// TIA Portal V15.1 export
// export: Created 2024-06-21T08:41:12.3335772Z, ExportSetting WithDefaults, DisplayName Totally Integrated Automation Portal, DisplayVersion V15.1 Update 5, DisplayName TIA Portal Openness, DisplayVersion V15.1 Update 5, DisplayName SINAMICS Startdrive Advanced, DisplayVersion V15.1, DisplayName G130, G150, S120, S150, SINAMICS MV, S210, DisplayVersion V15.1, DisplayName G110M, G120, G120C, G120D, G120P, DisplayVersion V15.1, DisplayName STEP 7 Professional, DisplayVersion V15.1 Update 5, DisplayName STEP 7 Safety, DisplayVersion V15.1, DisplayName WinCC Professional, DisplayVersion V15.1 Update 5, DisplayName SIMATIC Visualization Architect, DisplayVersion V15.1
FUNCTION_BLOCK "LGBHMILed"   // FB6683, FBD
TITLE = LGBHMILed
{ S7_Optimized_Access := 'TRUE' }
VERSION : 0.1
// =============================================================================
// This module handles indication for Start, Alarm Reset.
// =============================================================================
// stored: AutoNumber false, IsIECCheckEnabled false, IsRetainMemResEnabled false, MemoryReserve 100, SetENOAutomatically False, UDAEnableTagReadback false
   VAR_INPUT
      I_SafetyAckReq { ExternalAccessible := 'False'; ExternalVisible := 'False'; ExternalWritable := 'False'} : Bool;   // Safety acknowledge required
      I_SafetyOk { ExternalAccessible := 'False'; ExternalVisible := 'False'; ExternalWritable := 'False'} : Bool;   // All Safety ok
      I_PowerOnReq { ExternalAccessible := 'False'; ExternalVisible := 'False'; ExternalWritable := 'False'} : Bool;   // Request for power on (fast blinking of blue lamp)
      I_ResetSafety { ExternalAccessible := 'False'; ExternalVisible := 'False'; ExternalWritable := 'False'} : Bool;   // Reset Safety Signal of the Safety Zone
      C_ZSLevel { ExternalAccessible := 'False'; ExternalVisible := 'False'; ExternalWritable := 'False'} : Bool;   // ZS level OP
      C_PLCLevel { ExternalAccessible := 'False'; ExternalVisible := 'False'; ExternalWritable := 'False'} : Bool;   // PLC level OP
   END_VAR
   VAR_OUTPUT
      O_StartPBInd { ExternalAccessible := 'False'; ExternalVisible := 'False'; ExternalWritable := 'False'} : Bool;   // Start PB indication
      O_AlarmResetPBInd { ExternalAccessible := 'False'; ExternalVisible := 'False'; ExternalWritable := 'False'} : Bool;   // Alarm Reset PB Indication
   END_VAR
   VAR_IN_OUT
      IO_ModesZM1 : "Modes";   // Modes ZM1
      IO_ModesZM2 : "Modes";   // Modes ZM2
      IO_ModesZM3 : "Modes";   // Modes ZM3
      IO_ModesZM4 : "Modes";   // Modes ZM4
      IO_ModesZM5 : "Modes";   // Modes ZM5
      IO_ModesZM6 : "Modes";   // Modes ZM6
      IO_ModesZM7 : "Modes";   // Modes ZM7
      IO_ModesZM8 : "Modes";   // Modes ZM8
      IO_ModesZM9 : "Modes";   // Modes ZM9
      IO_ModesZM10 : "Modes";   // Modes ZM10
      IO_ModesZM11 : "Modes";   // Modes ZM11
      IO_ModesZM12 : "Modes";   // Modes ZM12
      IO_ModesZM13 : "Modes";   // Modes ZM13
      IO_ModesZM14 : "Modes";   // Modes ZM14
      IO_ModesZM15 : "Modes";   // Modes ZM15
      IO_ModesZM16 : "Modes";   // Modes ZM16
   END_VAR
   VAR
      ZMAlarmABLampSteadyCondition { ExternalAccessible := 'False'; ExternalVisible := 'False'; ExternalWritable := 'False'} : Bool;   // Alarm conditions active
      ZSAlarmABLampSteadyCondition { ExternalAccessible := 'False'; ExternalVisible := 'False'; ExternalWritable := 'False'} : Bool;   // Alarm conditions active
      PLCAlarmABLampSteadyCondition { ExternalAccessible := 'False'; ExternalVisible := 'False'; ExternalWritable := 'False'} : Bool;   // Alarm conditions active
      ZMAlarmABAckReq { ExternalAccessible := 'False'; ExternalVisible := 'False'; ExternalWritable := 'False'} : Bool;   // Alarm AB acknowledgement required
      ZSAlarmABAckReq { ExternalAccessible := 'False'; ExternalVisible := 'False'; ExternalWritable := 'False'} : Bool;   // Alarm AB acknowledgement required
      PLCAlarmABAckReq { ExternalAccessible := 'False'; ExternalVisible := 'False'; ExternalWritable := 'False'} : Bool;   // Alarm AB acknowledgement required
      BlueLampBlinkingCond { ExternalAccessible := 'False'; ExternalVisible := 'False'; ExternalWritable := 'False'} : Bool;   // Blue lamp blinking condition
      Lamptest { ExternalAccessible := 'False'; ExternalVisible := 'False'; ExternalWritable := 'False'} : Bool;   // Lamptest selected alternating signal
      LamptestSteady { ExternalAccessible := 'False'; ExternalVisible := 'False'; ExternalWritable := 'False'} : Bool;   // Lamptest selected steady signal
      AutoSel { ExternalAccessible := 'False'; ExternalVisible := 'False'; ExternalWritable := 'False'} : Bool;   // Automatic mode selected
      AutoMode { ExternalAccessible := 'False'; ExternalVisible := 'False'; ExternalWritable := 'False'} : Bool;   // Automatic mode active
      StartPBInd { ExternalAccessible := 'False'; ExternalVisible := 'False'; ExternalWritable := 'False'} : Bool;   // Start PB indication
      AlarmResetPBInd { ExternalAccessible := 'False'; ExternalVisible := 'False'; ExternalWritable := 'False'} : Bool;   // Alarm Reset PB Indication
   END_VAR
BEGIN

REGION Network 1: **** 4.2 - Machine status - Calculated **** ZM level Alarm condition AB active
   // Alarm condition AB active
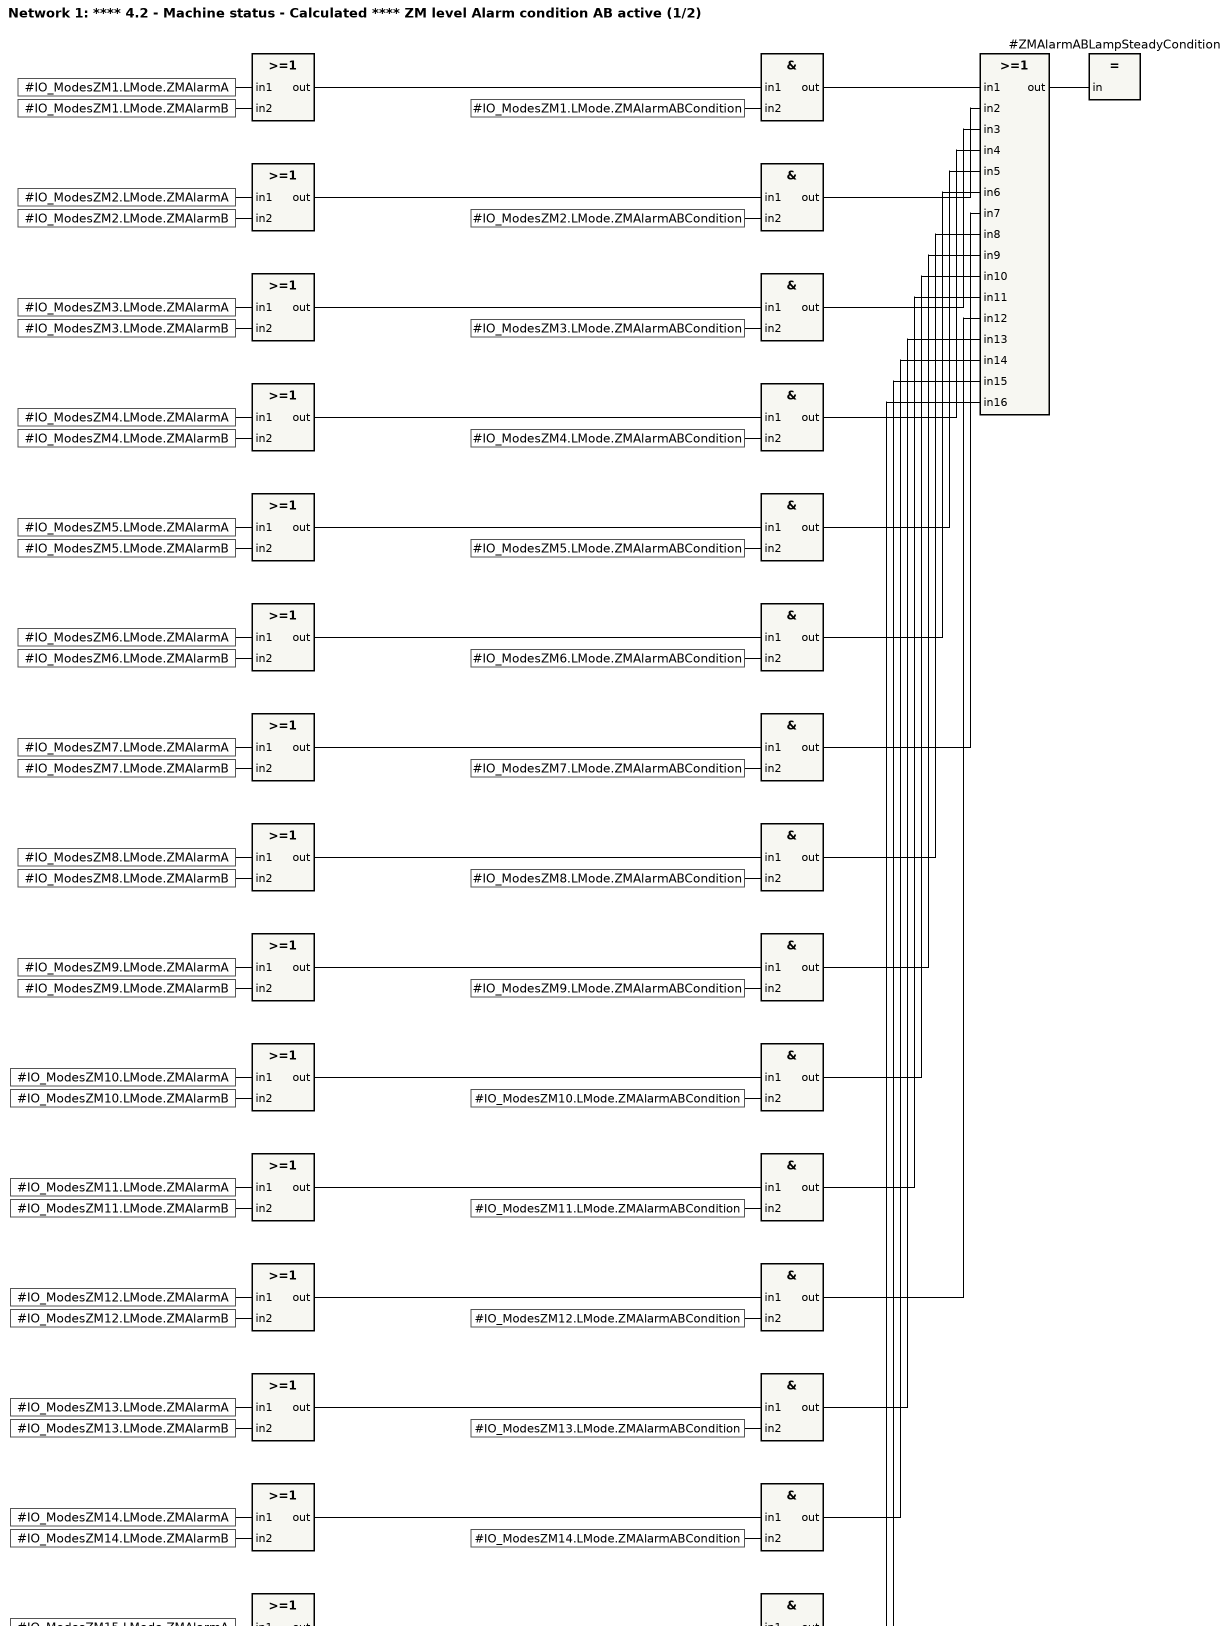
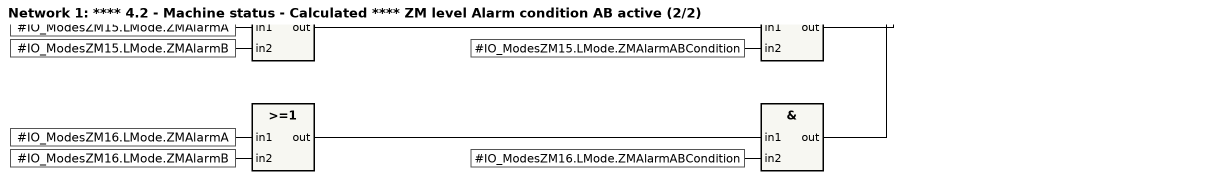
   #ZMAlarmABLampSteadyCondition := ((#IO_ModesZM1.LMode.ZMAlarmA OR #IO_ModesZM1.LMode.ZMAlarmB) AND #IO_ModesZM1.LMode.ZMAlarmABCondition) OR ((#IO_ModesZM2.LMode.ZMAlarmA OR #IO_ModesZM2.LMode.ZMAlarmB) AND #IO_ModesZM2.LMode.ZMAlarmABCondition) OR ((#IO_ModesZM3.LMode.ZMAlarmA OR #IO_ModesZM3.LMode.ZMAlarmB) AND #IO_ModesZM3.LMode.ZMAlarmABCondition) OR ((#IO_ModesZM4.LMode.ZMAlarmA OR #IO_ModesZM4.LMode.ZMAlarmB) AND #IO_ModesZM4.LMode.ZMAlarmABCondition) OR ((#IO_ModesZM5.LMode.ZMAlarmA OR #IO_ModesZM5.LMode.ZMAlarmB) AND #IO_ModesZM5.LMode.ZMAlarmABCondition) OR ((#IO_ModesZM6.LMode.ZMAlarmA OR #IO_ModesZM6.LMode.ZMAlarmB) AND #IO_ModesZM6.LMode.ZMAlarmABCondition) OR ((#IO_ModesZM7.LMode.ZMAlarmA OR #IO_ModesZM7.LMode.ZMAlarmB) AND #IO_ModesZM7.LMode.ZMAlarmABCondition) OR ((#IO_ModesZM8.LMode.ZMAlarmA OR #IO_ModesZM8.LMode.ZMAlarmB) AND #IO_ModesZM8.LMode.ZMAlarmABCondition) OR ((#IO_ModesZM9.LMode.ZMAlarmA OR #IO_ModesZM9.LMode.ZMAlarmB) AND #IO_ModesZM9.LMode.ZMAlarmABCondition) OR ((#IO_ModesZM10.LMode.ZMAlarmA OR #IO_ModesZM10.LMode.ZMAlarmB) AND #IO_ModesZM10.LMode.ZMAlarmABCondition) OR ((#IO_ModesZM11.LMode.ZMAlarmA OR #IO_ModesZM11.LMode.ZMAlarmB) AND #IO_ModesZM11.LMode.ZMAlarmABCondition) OR ((#IO_ModesZM12.LMode.ZMAlarmA OR #IO_ModesZM12.LMode.ZMAlarmB) AND #IO_ModesZM12.LMode.ZMAlarmABCondition) OR ((#IO_ModesZM13.LMode.ZMAlarmA OR #IO_ModesZM13.LMode.ZMAlarmB) AND #IO_ModesZM13.LMode.ZMAlarmABCondition) OR ((#IO_ModesZM14.LMode.ZMAlarmA OR #IO_ModesZM14.LMode.ZMAlarmB) AND #IO_ModesZM14.LMode.ZMAlarmABCondition) OR ((#IO_ModesZM15.LMode.ZMAlarmA OR #IO_ModesZM15.LMode.ZMAlarmB) AND #IO_ModesZM15.LMode.ZMAlarmABCondition) OR ((#IO_ModesZM16.LMode.ZMAlarmA OR #IO_ModesZM16.LMode.ZMAlarmB) AND #IO_ModesZM16.LMode.ZMAlarmABCondition);
END_REGION

REGION Network 2: **** 4.2 - Machine status - Calculated **** ZS level Alarm condition AB active
   // Alarm condition AB active
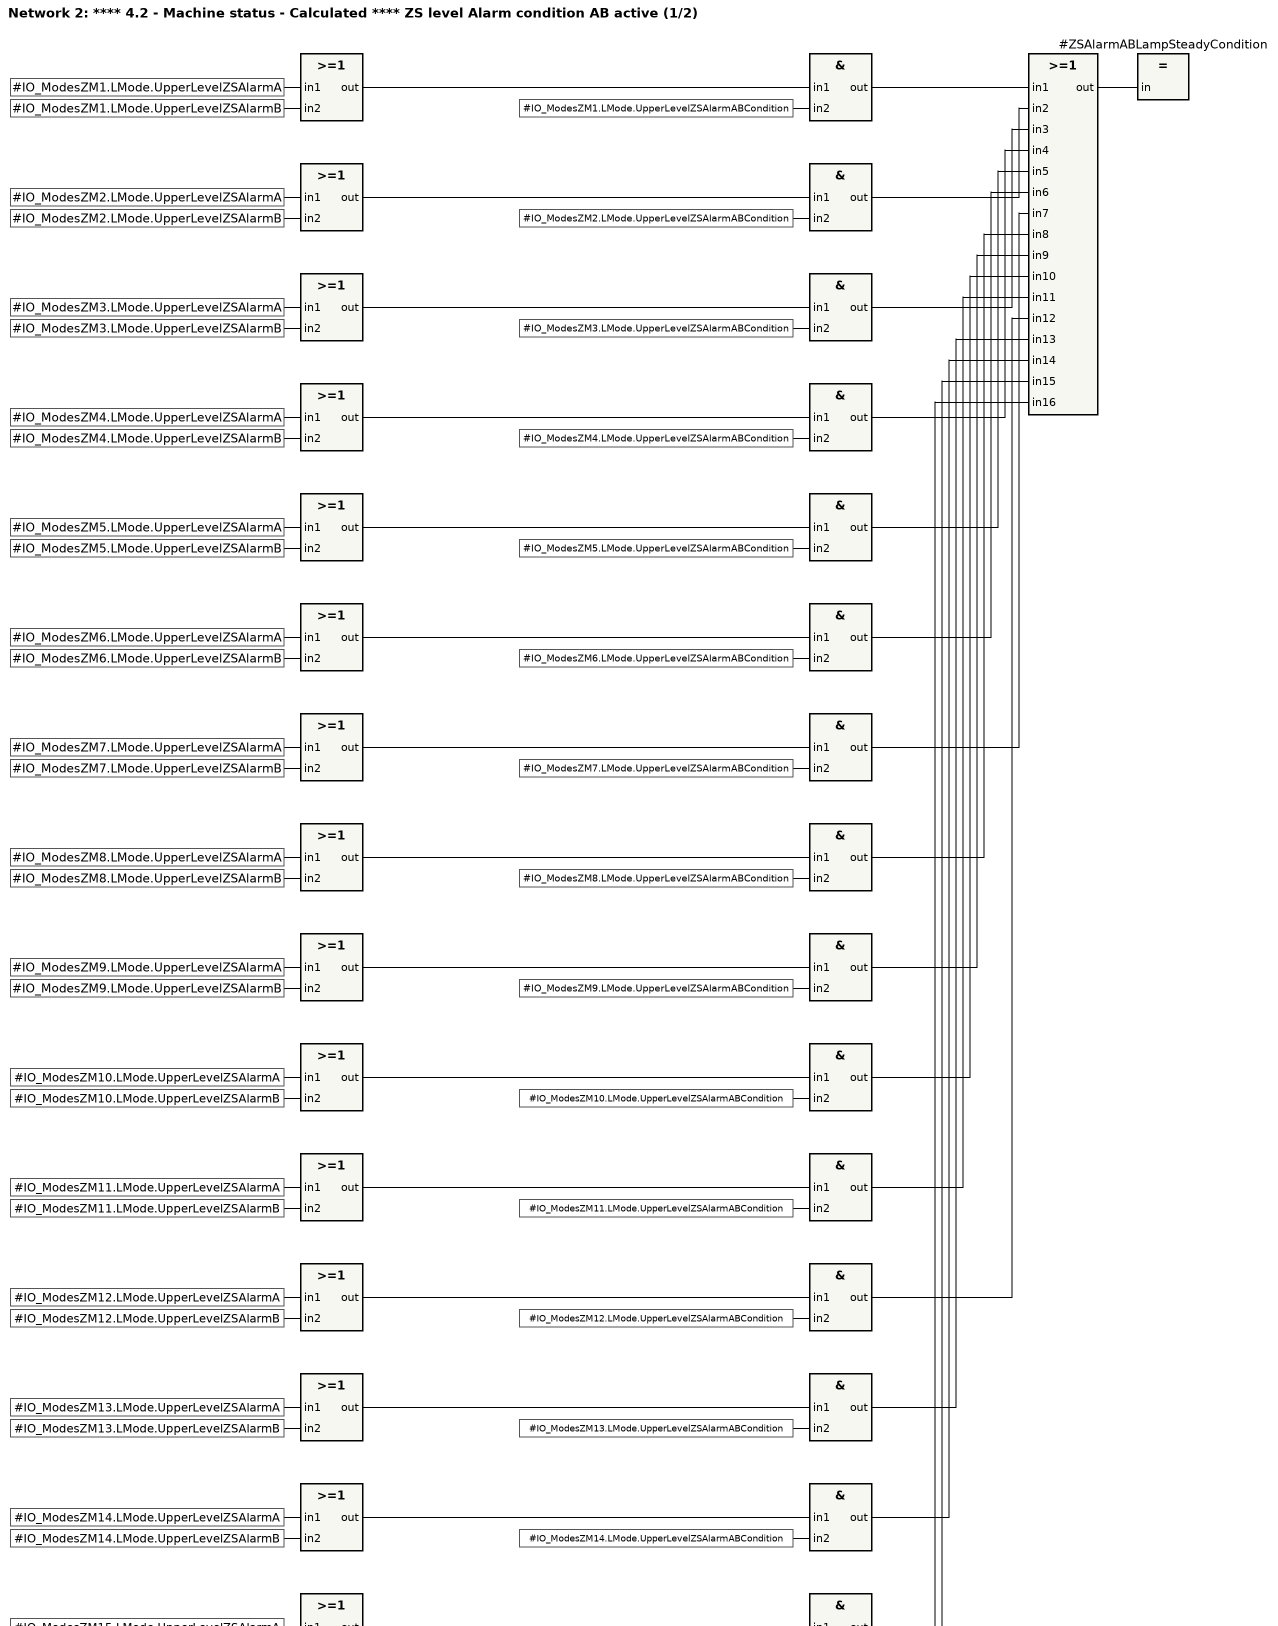
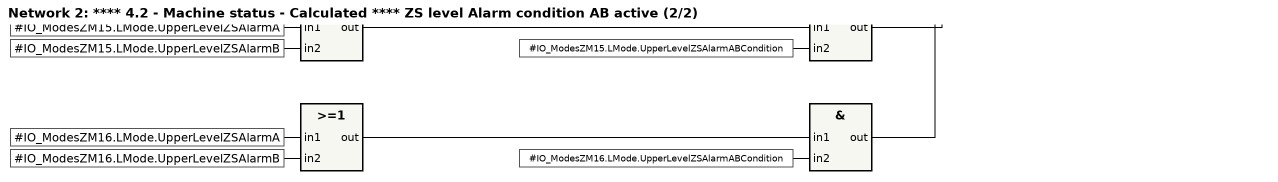
   #ZSAlarmABLampSteadyCondition := ((#IO_ModesZM1.LMode.UpperLevelZSAlarmA OR #IO_ModesZM1.LMode.UpperLevelZSAlarmB) AND #IO_ModesZM1.LMode.UpperLevelZSAlarmABCondition) OR ((#IO_ModesZM2.LMode.UpperLevelZSAlarmA OR #IO_ModesZM2.LMode.UpperLevelZSAlarmB) AND #IO_ModesZM2.LMode.UpperLevelZSAlarmABCondition) OR ((#IO_ModesZM3.LMode.UpperLevelZSAlarmA OR #IO_ModesZM3.LMode.UpperLevelZSAlarmB) AND #IO_ModesZM3.LMode.UpperLevelZSAlarmABCondition) OR ((#IO_ModesZM4.LMode.UpperLevelZSAlarmA OR #IO_ModesZM4.LMode.UpperLevelZSAlarmB) AND #IO_ModesZM4.LMode.UpperLevelZSAlarmABCondition) OR ((#IO_ModesZM5.LMode.UpperLevelZSAlarmA OR #IO_ModesZM5.LMode.UpperLevelZSAlarmB) AND #IO_ModesZM5.LMode.UpperLevelZSAlarmABCondition) OR ((#IO_ModesZM6.LMode.UpperLevelZSAlarmA OR #IO_ModesZM6.LMode.UpperLevelZSAlarmB) AND #IO_ModesZM6.LMode.UpperLevelZSAlarmABCondition) OR ((#IO_ModesZM7.LMode.UpperLevelZSAlarmA OR #IO_ModesZM7.LMode.UpperLevelZSAlarmB) AND #IO_ModesZM7.LMode.UpperLevelZSAlarmABCondition) OR ((#IO_ModesZM8.LMode.UpperLevelZSAlarmA OR #IO_ModesZM8.LMode.UpperLevelZSAlarmB) AND #IO_ModesZM8.LMode.UpperLevelZSAlarmABCondition) OR ((#IO_ModesZM9.LMode.UpperLevelZSAlarmA OR #IO_ModesZM9.LMode.UpperLevelZSAlarmB) AND #IO_ModesZM9.LMode.UpperLevelZSAlarmABCondition) OR ((#IO_ModesZM10.LMode.UpperLevelZSAlarmA OR #IO_ModesZM10.LMode.UpperLevelZSAlarmB) AND #IO_ModesZM10.LMode.UpperLevelZSAlarmABCondition) OR ((#IO_ModesZM11.LMode.UpperLevelZSAlarmA OR #IO_ModesZM11.LMode.UpperLevelZSAlarmB) AND #IO_ModesZM11.LMode.UpperLevelZSAlarmABCondition) OR ((#IO_ModesZM12.LMode.UpperLevelZSAlarmA OR #IO_ModesZM12.LMode.UpperLevelZSAlarmB) AND #IO_ModesZM12.LMode.UpperLevelZSAlarmABCondition) OR ((#IO_ModesZM13.LMode.UpperLevelZSAlarmA OR #IO_ModesZM13.LMode.UpperLevelZSAlarmB) AND #IO_ModesZM13.LMode.UpperLevelZSAlarmABCondition) OR ((#IO_ModesZM14.LMode.UpperLevelZSAlarmA OR #IO_ModesZM14.LMode.UpperLevelZSAlarmB) AND #IO_ModesZM14.LMode.UpperLevelZSAlarmABCondition) OR ((#IO_ModesZM15.LMode.UpperLevelZSAlarmA OR #IO_ModesZM15.LMode.UpperLevelZSAlarmB) AND #IO_ModesZM15.LMode.UpperLevelZSAlarmABCondition) OR ((#IO_ModesZM16.LMode.UpperLevelZSAlarmA OR #IO_ModesZM16.LMode.UpperLevelZSAlarmB) AND #IO_ModesZM16.LMode.UpperLevelZSAlarmABCondition);
END_REGION

REGION Network 3: **** 4.2 - Machine status - Calculated **** PLC level Alarm condition AB active
   // Alarm condition AB active
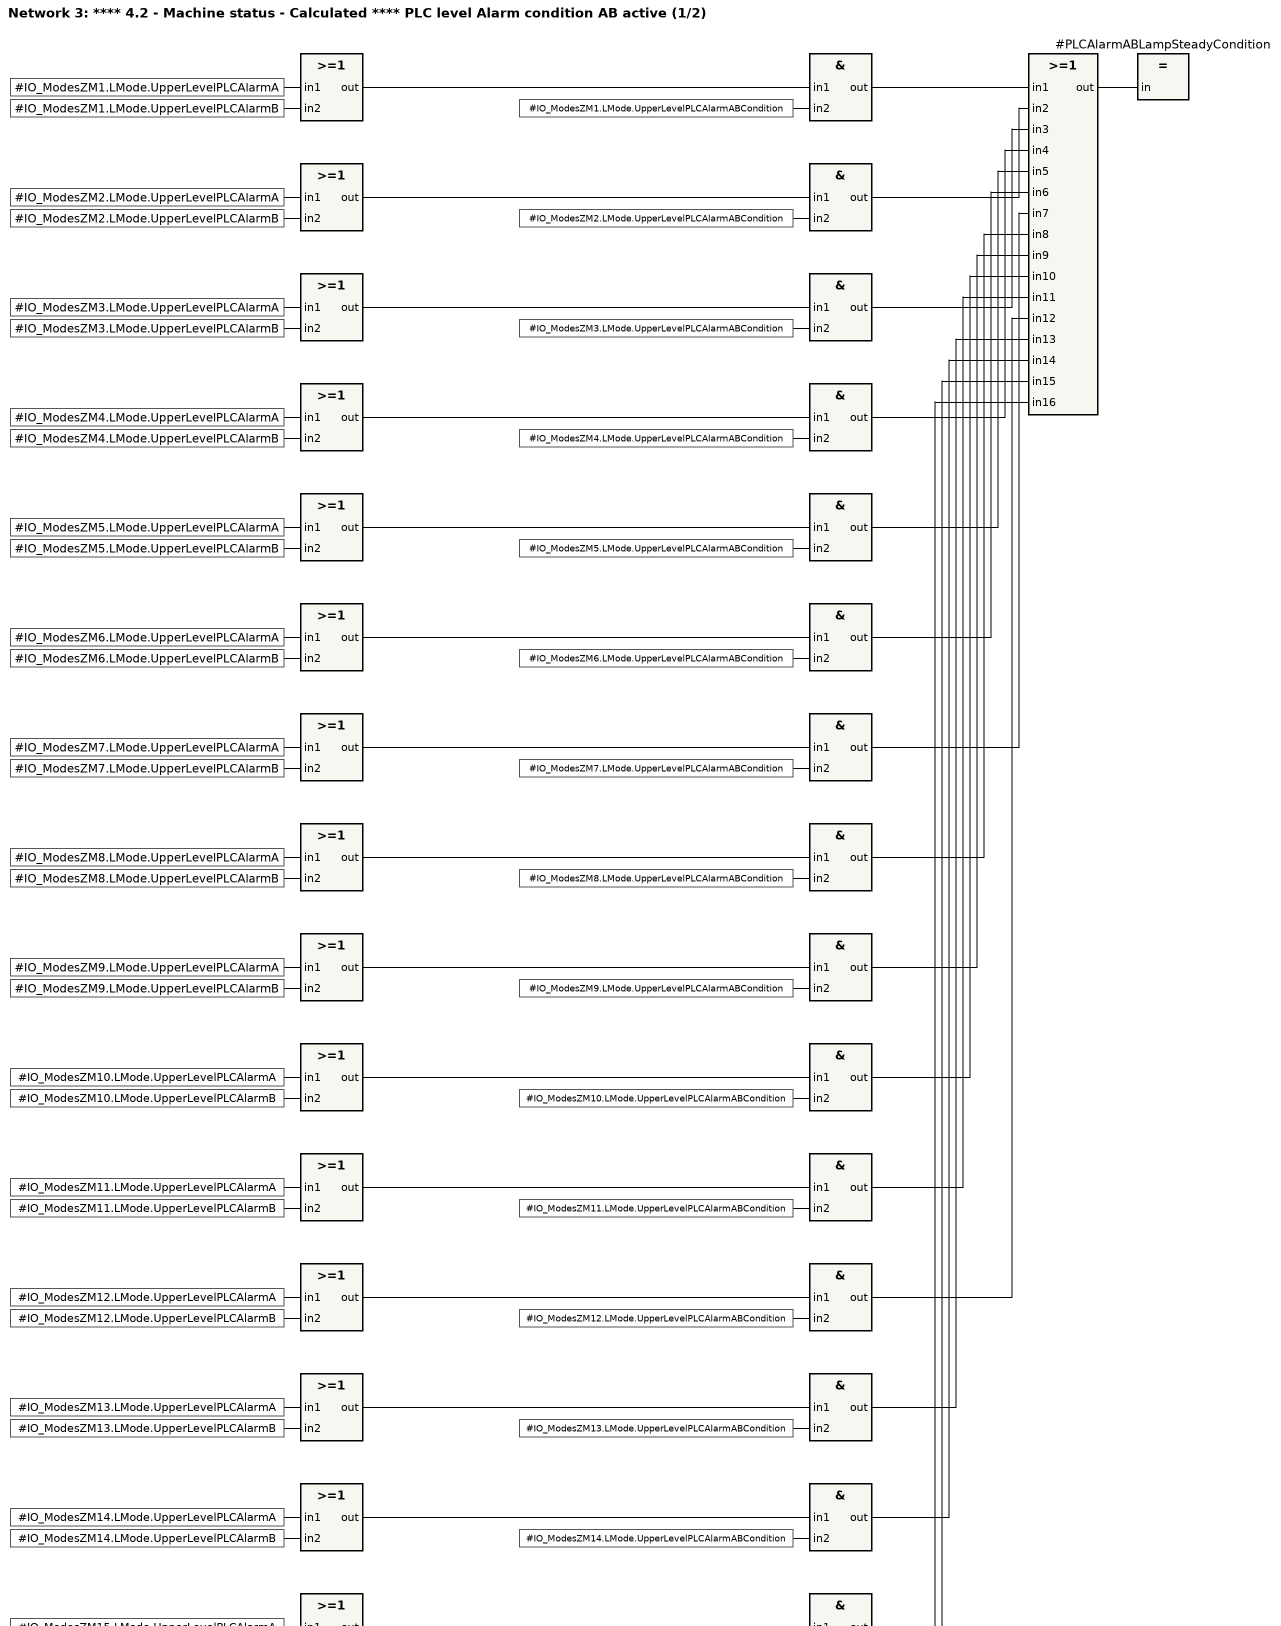
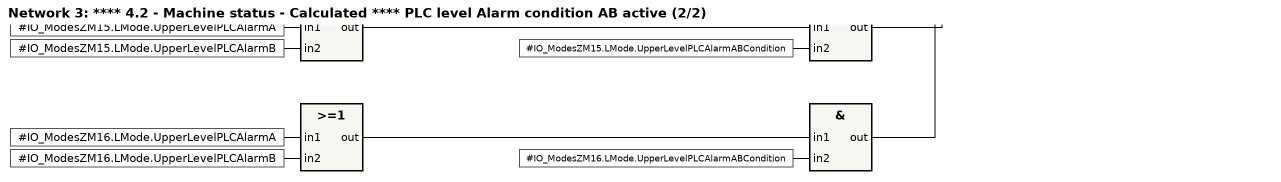
   #PLCAlarmABLampSteadyCondition := ((#IO_ModesZM1.LMode.UpperLevelPLCAlarmA OR #IO_ModesZM1.LMode.UpperLevelPLCAlarmB) AND #IO_ModesZM1.LMode.UpperLevelPLCAlarmABCondition) OR ((#IO_ModesZM2.LMode.UpperLevelPLCAlarmA OR #IO_ModesZM2.LMode.UpperLevelPLCAlarmB) AND #IO_ModesZM2.LMode.UpperLevelPLCAlarmABCondition) OR ((#IO_ModesZM3.LMode.UpperLevelPLCAlarmA OR #IO_ModesZM3.LMode.UpperLevelPLCAlarmB) AND #IO_ModesZM3.LMode.UpperLevelPLCAlarmABCondition) OR ((#IO_ModesZM4.LMode.UpperLevelPLCAlarmA OR #IO_ModesZM4.LMode.UpperLevelPLCAlarmB) AND #IO_ModesZM4.LMode.UpperLevelPLCAlarmABCondition) OR ((#IO_ModesZM5.LMode.UpperLevelPLCAlarmA OR #IO_ModesZM5.LMode.UpperLevelPLCAlarmB) AND #IO_ModesZM5.LMode.UpperLevelPLCAlarmABCondition) OR ((#IO_ModesZM6.LMode.UpperLevelPLCAlarmA OR #IO_ModesZM6.LMode.UpperLevelPLCAlarmB) AND #IO_ModesZM6.LMode.UpperLevelPLCAlarmABCondition) OR ((#IO_ModesZM7.LMode.UpperLevelPLCAlarmA OR #IO_ModesZM7.LMode.UpperLevelPLCAlarmB) AND #IO_ModesZM7.LMode.UpperLevelPLCAlarmABCondition) OR ((#IO_ModesZM8.LMode.UpperLevelPLCAlarmA OR #IO_ModesZM8.LMode.UpperLevelPLCAlarmB) AND #IO_ModesZM8.LMode.UpperLevelPLCAlarmABCondition) OR ((#IO_ModesZM9.LMode.UpperLevelPLCAlarmA OR #IO_ModesZM9.LMode.UpperLevelPLCAlarmB) AND #IO_ModesZM9.LMode.UpperLevelPLCAlarmABCondition) OR ((#IO_ModesZM10.LMode.UpperLevelPLCAlarmA OR #IO_ModesZM10.LMode.UpperLevelPLCAlarmB) AND #IO_ModesZM10.LMode.UpperLevelPLCAlarmABCondition) OR ((#IO_ModesZM11.LMode.UpperLevelPLCAlarmA OR #IO_ModesZM11.LMode.UpperLevelPLCAlarmB) AND #IO_ModesZM11.LMode.UpperLevelPLCAlarmABCondition) OR ((#IO_ModesZM12.LMode.UpperLevelPLCAlarmA OR #IO_ModesZM12.LMode.UpperLevelPLCAlarmB) AND #IO_ModesZM12.LMode.UpperLevelPLCAlarmABCondition) OR ((#IO_ModesZM13.LMode.UpperLevelPLCAlarmA OR #IO_ModesZM13.LMode.UpperLevelPLCAlarmB) AND #IO_ModesZM13.LMode.UpperLevelPLCAlarmABCondition) OR ((#IO_ModesZM14.LMode.UpperLevelPLCAlarmA OR #IO_ModesZM14.LMode.UpperLevelPLCAlarmB) AND #IO_ModesZM14.LMode.UpperLevelPLCAlarmABCondition) OR ((#IO_ModesZM15.LMode.UpperLevelPLCAlarmA OR #IO_ModesZM15.LMode.UpperLevelPLCAlarmB) AND #IO_ModesZM15.LMode.UpperLevelPLCAlarmABCondition) OR ((#IO_ModesZM16.LMode.UpperLevelPLCAlarmA OR #IO_ModesZM16.LMode.UpperLevelPLCAlarmB) AND #IO_ModesZM16.LMode.UpperLevelPLCAlarmABCondition);
END_REGION

REGION Network 4: **** 4.2 - Machine status - Calculated **** ZM level Alarm AB Acknowledge Request
   // Alarm AB Acknowledge Request
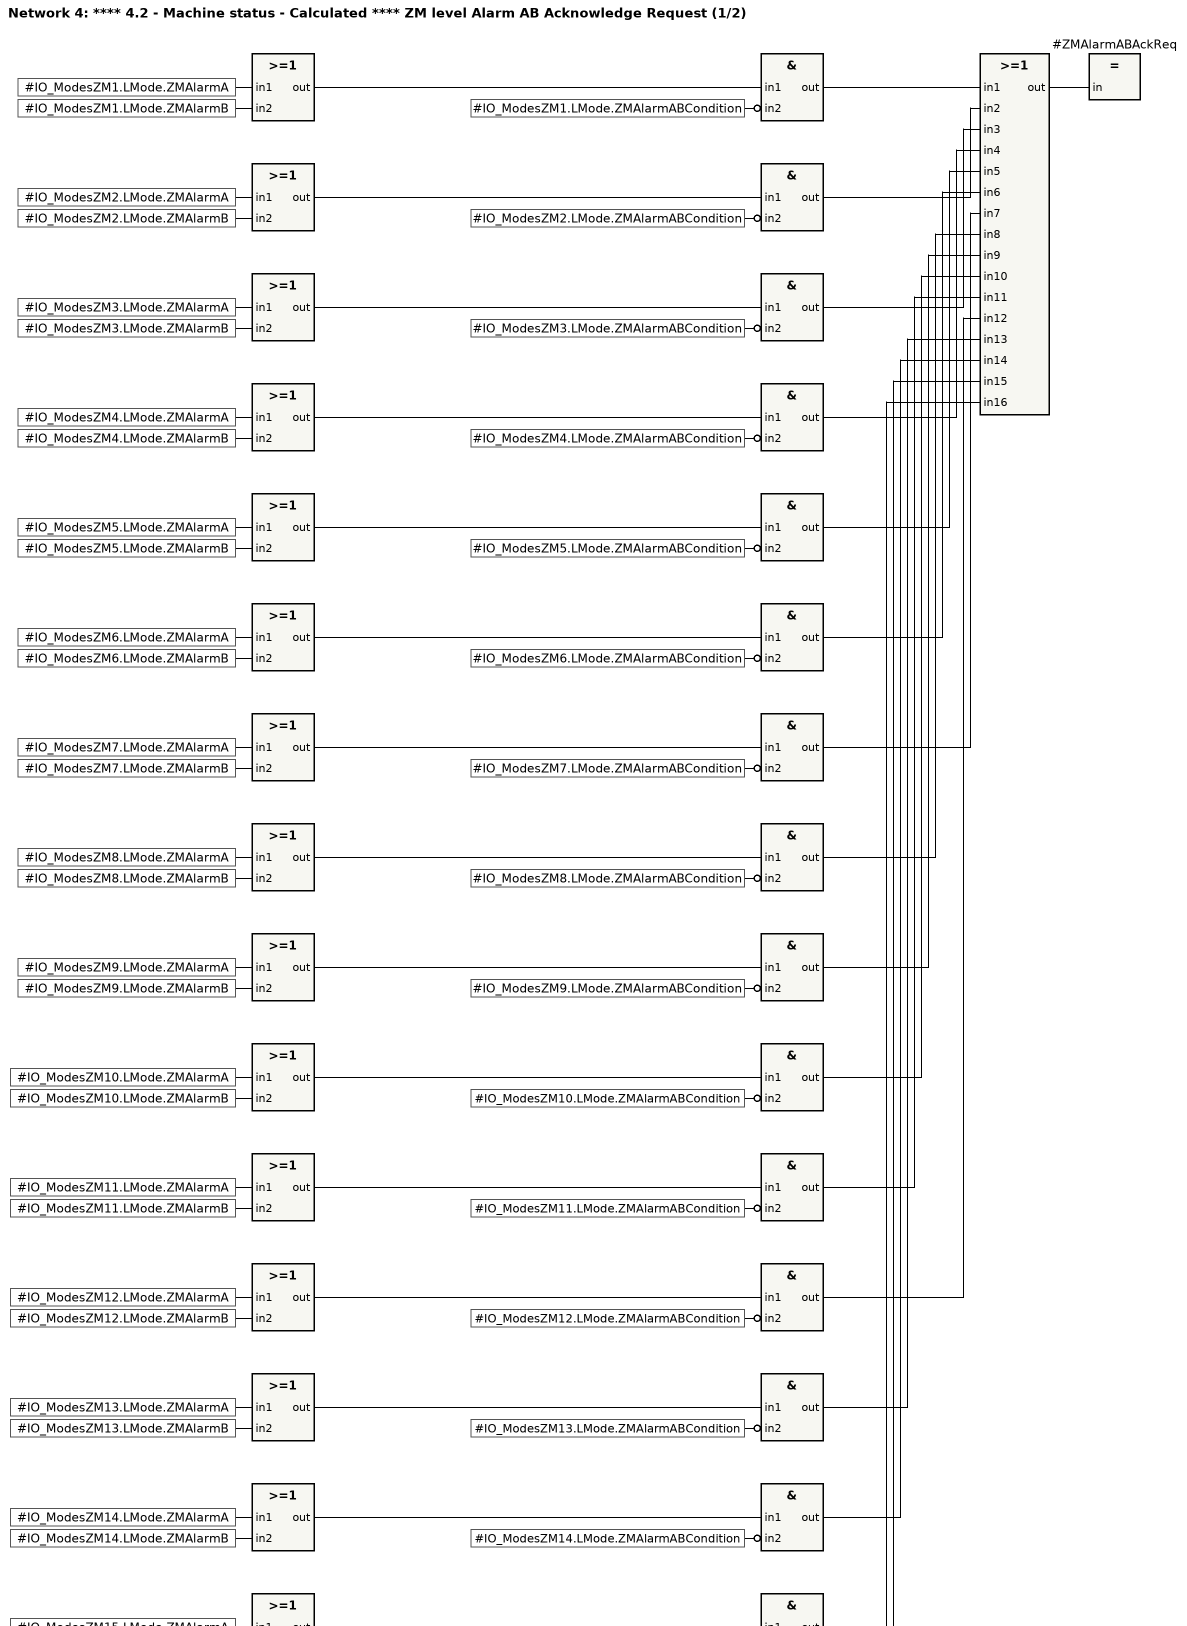
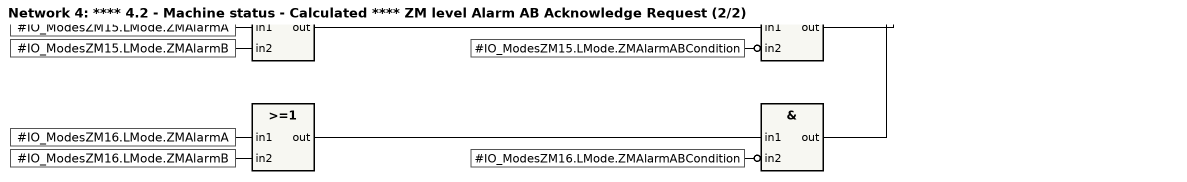
   #ZMAlarmABAckReq := ((#IO_ModesZM1.LMode.ZMAlarmA OR #IO_ModesZM1.LMode.ZMAlarmB) AND NOT #IO_ModesZM1.LMode.ZMAlarmABCondition) OR ((#IO_ModesZM2.LMode.ZMAlarmA OR #IO_ModesZM2.LMode.ZMAlarmB) AND NOT #IO_ModesZM2.LMode.ZMAlarmABCondition) OR ((#IO_ModesZM3.LMode.ZMAlarmA OR #IO_ModesZM3.LMode.ZMAlarmB) AND NOT #IO_ModesZM3.LMode.ZMAlarmABCondition) OR ((#IO_ModesZM4.LMode.ZMAlarmA OR #IO_ModesZM4.LMode.ZMAlarmB) AND NOT #IO_ModesZM4.LMode.ZMAlarmABCondition) OR ((#IO_ModesZM5.LMode.ZMAlarmA OR #IO_ModesZM5.LMode.ZMAlarmB) AND NOT #IO_ModesZM5.LMode.ZMAlarmABCondition) OR ((#IO_ModesZM6.LMode.ZMAlarmA OR #IO_ModesZM6.LMode.ZMAlarmB) AND NOT #IO_ModesZM6.LMode.ZMAlarmABCondition) OR ((#IO_ModesZM7.LMode.ZMAlarmA OR #IO_ModesZM7.LMode.ZMAlarmB) AND NOT #IO_ModesZM7.LMode.ZMAlarmABCondition) OR ((#IO_ModesZM8.LMode.ZMAlarmA OR #IO_ModesZM8.LMode.ZMAlarmB) AND NOT #IO_ModesZM8.LMode.ZMAlarmABCondition) OR ((#IO_ModesZM9.LMode.ZMAlarmA OR #IO_ModesZM9.LMode.ZMAlarmB) AND NOT #IO_ModesZM9.LMode.ZMAlarmABCondition) OR ((#IO_ModesZM10.LMode.ZMAlarmA OR #IO_ModesZM10.LMode.ZMAlarmB) AND NOT #IO_ModesZM10.LMode.ZMAlarmABCondition) OR ((#IO_ModesZM11.LMode.ZMAlarmA OR #IO_ModesZM11.LMode.ZMAlarmB) AND NOT #IO_ModesZM11.LMode.ZMAlarmABCondition) OR ((#IO_ModesZM12.LMode.ZMAlarmA OR #IO_ModesZM12.LMode.ZMAlarmB) AND NOT #IO_ModesZM12.LMode.ZMAlarmABCondition) OR ((#IO_ModesZM13.LMode.ZMAlarmA OR #IO_ModesZM13.LMode.ZMAlarmB) AND NOT #IO_ModesZM13.LMode.ZMAlarmABCondition) OR ((#IO_ModesZM14.LMode.ZMAlarmA OR #IO_ModesZM14.LMode.ZMAlarmB) AND NOT #IO_ModesZM14.LMode.ZMAlarmABCondition) OR ((#IO_ModesZM15.LMode.ZMAlarmA OR #IO_ModesZM15.LMode.ZMAlarmB) AND NOT #IO_ModesZM15.LMode.ZMAlarmABCondition) OR ((#IO_ModesZM16.LMode.ZMAlarmA OR #IO_ModesZM16.LMode.ZMAlarmB) AND NOT #IO_ModesZM16.LMode.ZMAlarmABCondition);
END_REGION

REGION Network 5: **** 4.2 - Machine status - Calculated **** ZS level Alarm AB Acknowledge Request
   // Alarm AB Acknowledge Request
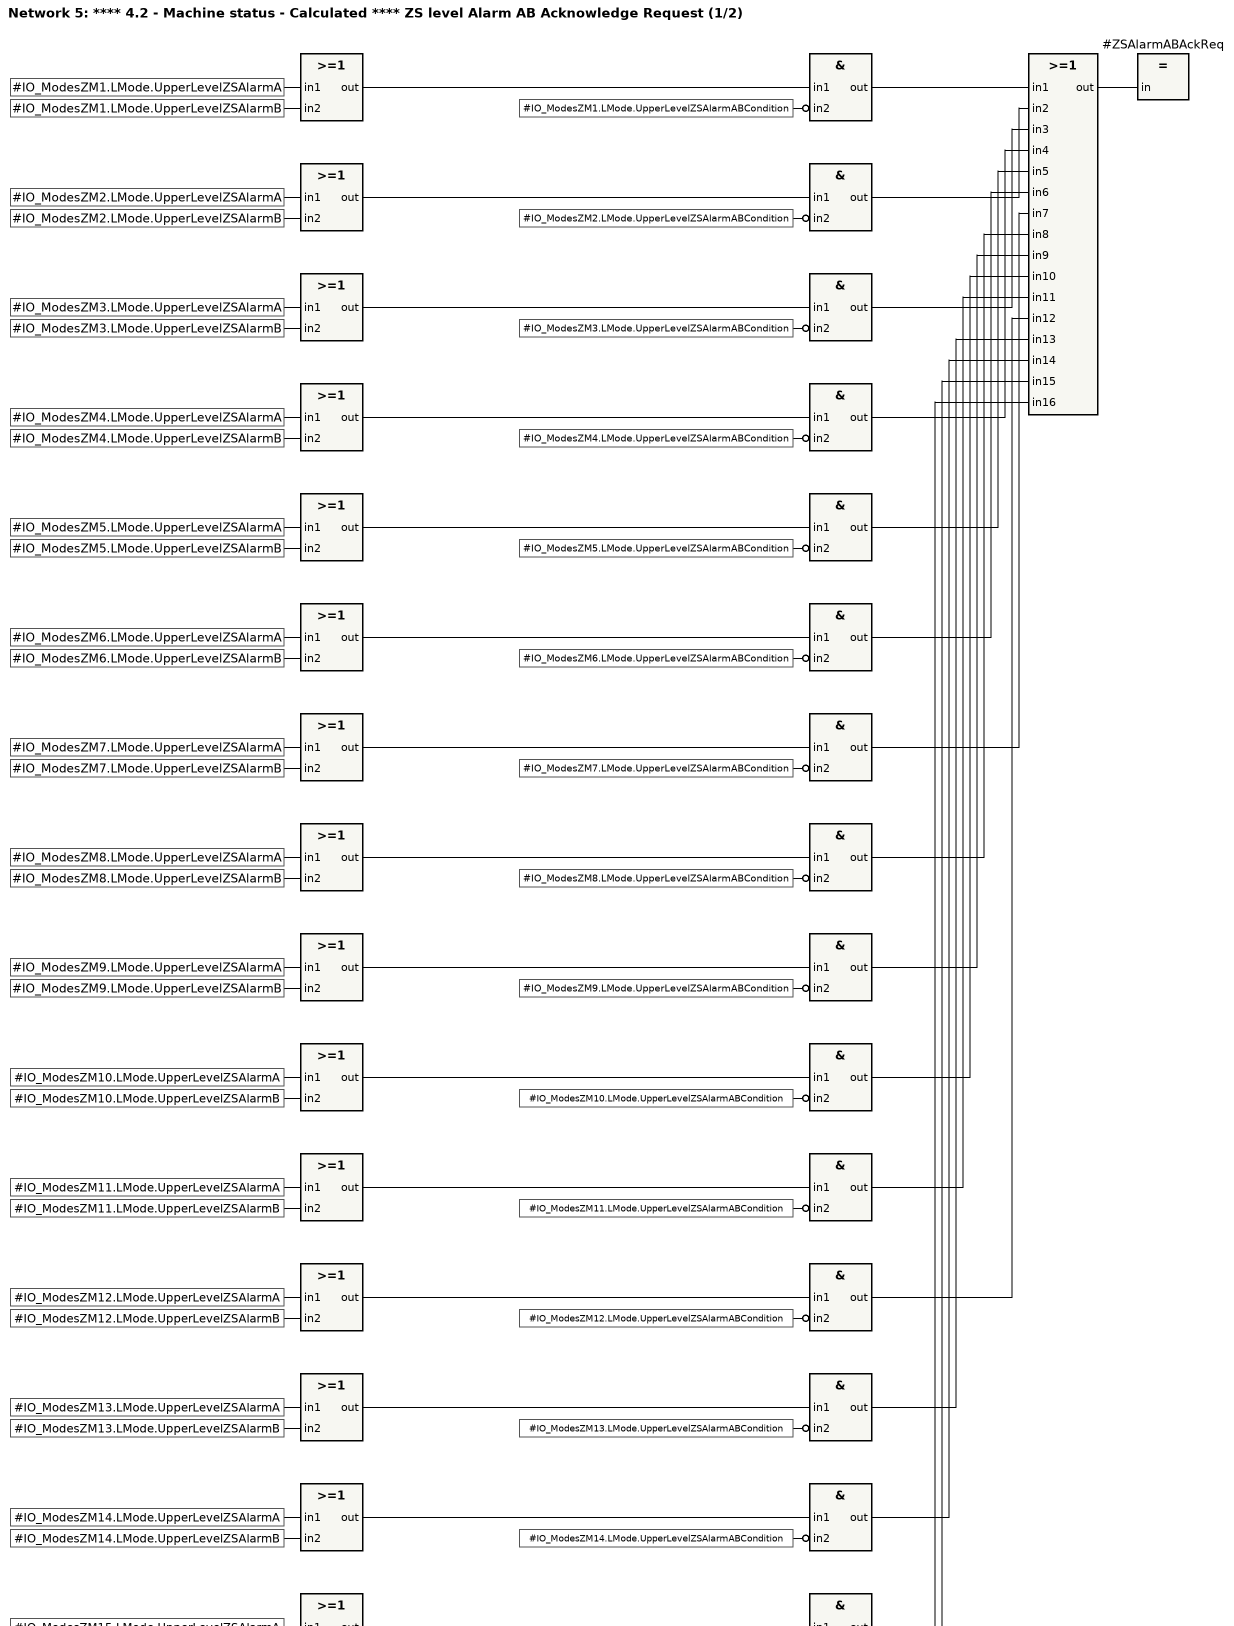
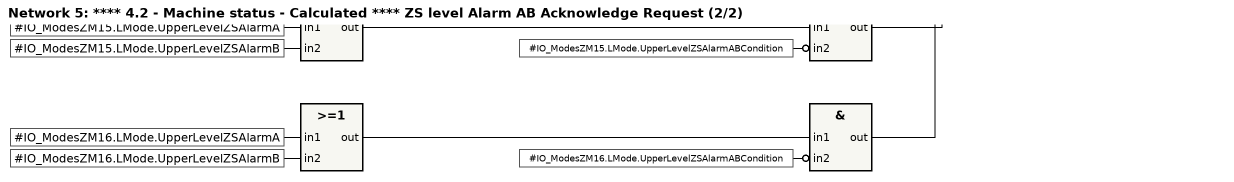
   #ZSAlarmABAckReq := ((#IO_ModesZM1.LMode.UpperLevelZSAlarmA OR #IO_ModesZM1.LMode.UpperLevelZSAlarmB) AND NOT #IO_ModesZM1.LMode.UpperLevelZSAlarmABCondition) OR ((#IO_ModesZM2.LMode.UpperLevelZSAlarmA OR #IO_ModesZM2.LMode.UpperLevelZSAlarmB) AND NOT #IO_ModesZM2.LMode.UpperLevelZSAlarmABCondition) OR ((#IO_ModesZM3.LMode.UpperLevelZSAlarmA OR #IO_ModesZM3.LMode.UpperLevelZSAlarmB) AND NOT #IO_ModesZM3.LMode.UpperLevelZSAlarmABCondition) OR ((#IO_ModesZM4.LMode.UpperLevelZSAlarmA OR #IO_ModesZM4.LMode.UpperLevelZSAlarmB) AND NOT #IO_ModesZM4.LMode.UpperLevelZSAlarmABCondition) OR ((#IO_ModesZM5.LMode.UpperLevelZSAlarmA OR #IO_ModesZM5.LMode.UpperLevelZSAlarmB) AND NOT #IO_ModesZM5.LMode.UpperLevelZSAlarmABCondition) OR ((#IO_ModesZM6.LMode.UpperLevelZSAlarmA OR #IO_ModesZM6.LMode.UpperLevelZSAlarmB) AND NOT #IO_ModesZM6.LMode.UpperLevelZSAlarmABCondition) OR ((#IO_ModesZM7.LMode.UpperLevelZSAlarmA OR #IO_ModesZM7.LMode.UpperLevelZSAlarmB) AND NOT #IO_ModesZM7.LMode.UpperLevelZSAlarmABCondition) OR ((#IO_ModesZM8.LMode.UpperLevelZSAlarmA OR #IO_ModesZM8.LMode.UpperLevelZSAlarmB) AND NOT #IO_ModesZM8.LMode.UpperLevelZSAlarmABCondition) OR ((#IO_ModesZM9.LMode.UpperLevelZSAlarmA OR #IO_ModesZM9.LMode.UpperLevelZSAlarmB) AND NOT #IO_ModesZM9.LMode.UpperLevelZSAlarmABCondition) OR ((#IO_ModesZM10.LMode.UpperLevelZSAlarmA OR #IO_ModesZM10.LMode.UpperLevelZSAlarmB) AND NOT #IO_ModesZM10.LMode.UpperLevelZSAlarmABCondition) OR ((#IO_ModesZM11.LMode.UpperLevelZSAlarmA OR #IO_ModesZM11.LMode.UpperLevelZSAlarmB) AND NOT #IO_ModesZM11.LMode.UpperLevelZSAlarmABCondition) OR ((#IO_ModesZM12.LMode.UpperLevelZSAlarmA OR #IO_ModesZM12.LMode.UpperLevelZSAlarmB) AND NOT #IO_ModesZM12.LMode.UpperLevelZSAlarmABCondition) OR ((#IO_ModesZM13.LMode.UpperLevelZSAlarmA OR #IO_ModesZM13.LMode.UpperLevelZSAlarmB) AND NOT #IO_ModesZM13.LMode.UpperLevelZSAlarmABCondition) OR ((#IO_ModesZM14.LMode.UpperLevelZSAlarmA OR #IO_ModesZM14.LMode.UpperLevelZSAlarmB) AND NOT #IO_ModesZM14.LMode.UpperLevelZSAlarmABCondition) OR ((#IO_ModesZM15.LMode.UpperLevelZSAlarmA OR #IO_ModesZM15.LMode.UpperLevelZSAlarmB) AND NOT #IO_ModesZM15.LMode.UpperLevelZSAlarmABCondition) OR ((#IO_ModesZM16.LMode.UpperLevelZSAlarmA OR #IO_ModesZM16.LMode.UpperLevelZSAlarmB) AND NOT #IO_ModesZM16.LMode.UpperLevelZSAlarmABCondition);
END_REGION

REGION Network 6: **** 4.2 - Machine status - Calculated **** PLC level Alarm AB Acknowledge Request
   // Alarm AB Acknowledge Request
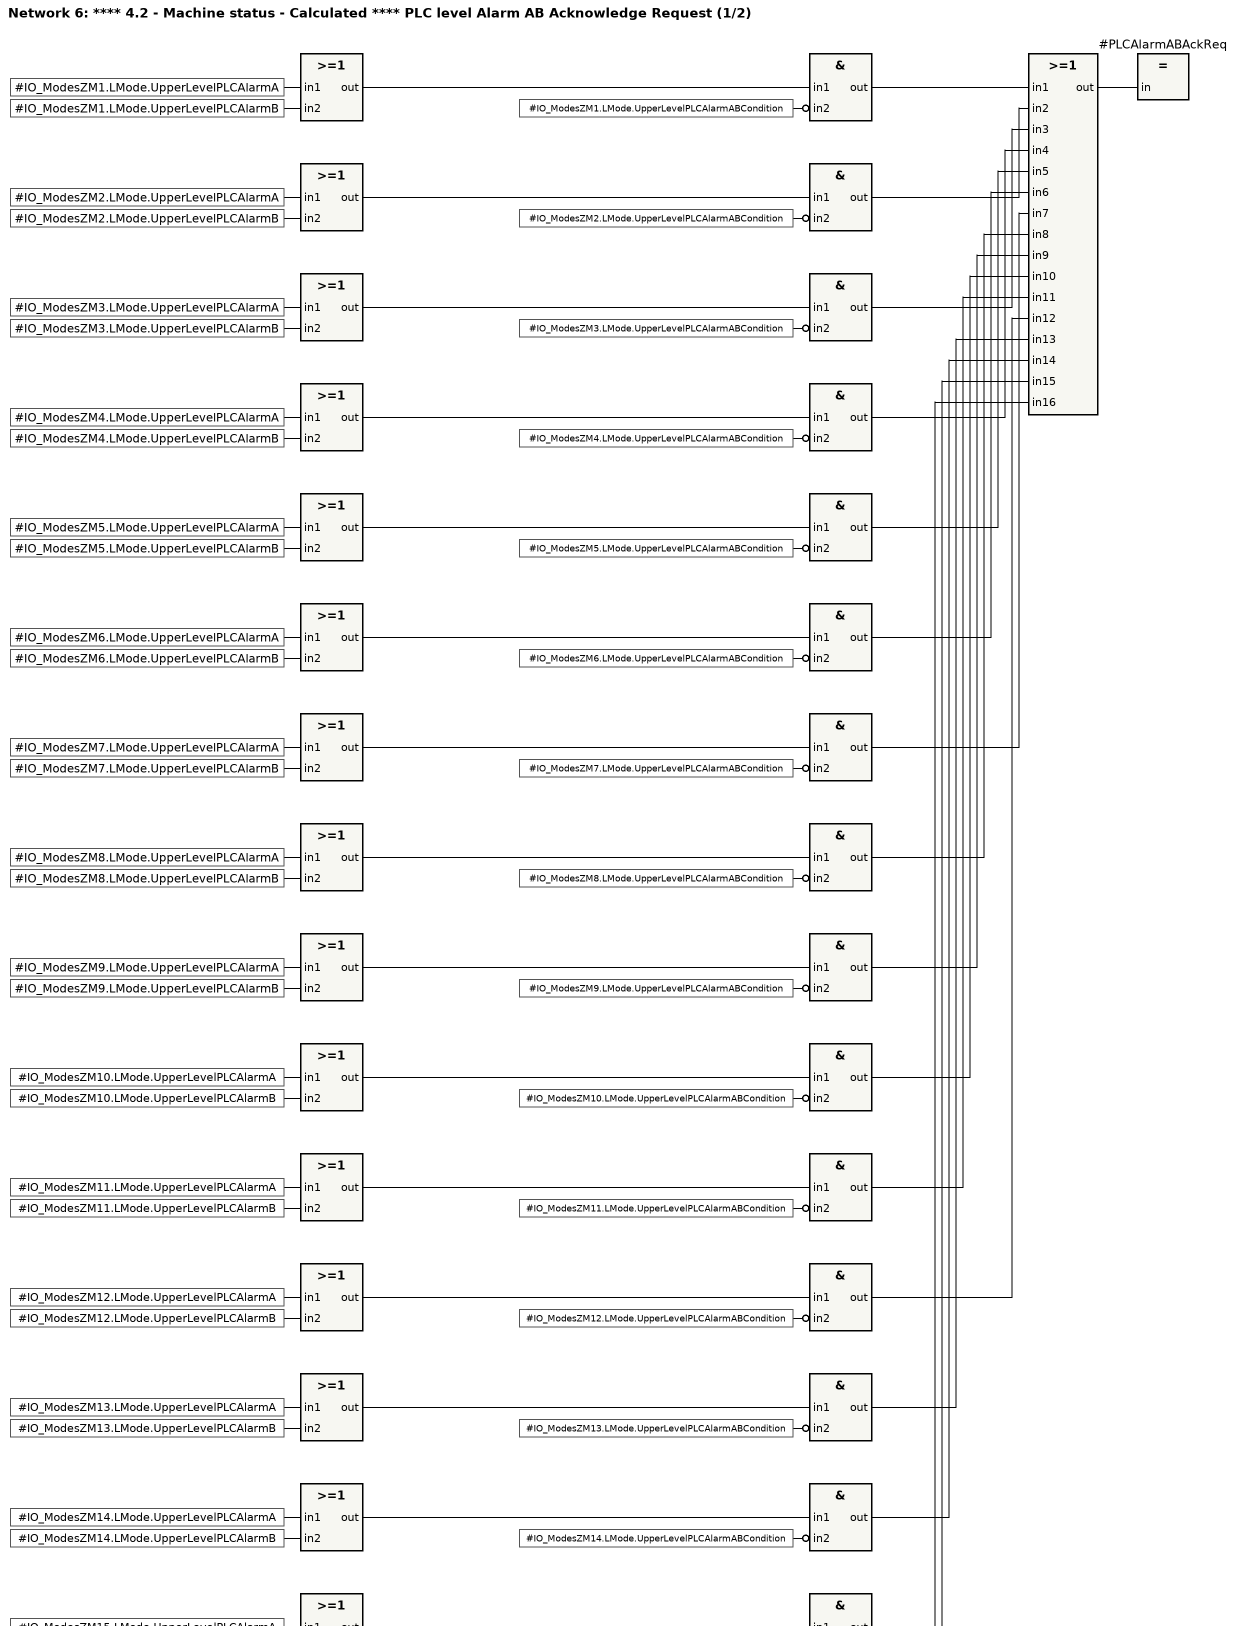
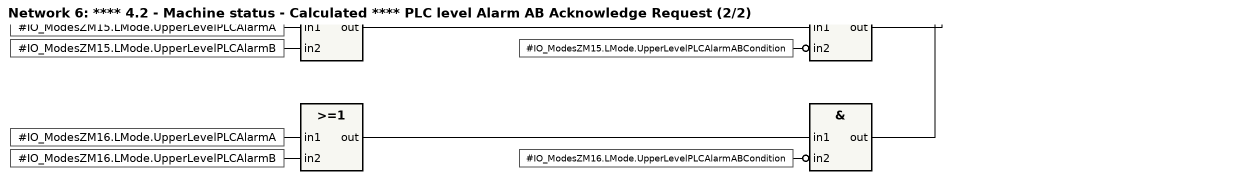
   #PLCAlarmABAckReq := ((#IO_ModesZM1.LMode.UpperLevelPLCAlarmA OR #IO_ModesZM1.LMode.UpperLevelPLCAlarmB) AND NOT #IO_ModesZM1.LMode.UpperLevelPLCAlarmABCondition) OR ((#IO_ModesZM2.LMode.UpperLevelPLCAlarmA OR #IO_ModesZM2.LMode.UpperLevelPLCAlarmB) AND NOT #IO_ModesZM2.LMode.UpperLevelPLCAlarmABCondition) OR ((#IO_ModesZM3.LMode.UpperLevelPLCAlarmA OR #IO_ModesZM3.LMode.UpperLevelPLCAlarmB) AND NOT #IO_ModesZM3.LMode.UpperLevelPLCAlarmABCondition) OR ((#IO_ModesZM4.LMode.UpperLevelPLCAlarmA OR #IO_ModesZM4.LMode.UpperLevelPLCAlarmB) AND NOT #IO_ModesZM4.LMode.UpperLevelPLCAlarmABCondition) OR ((#IO_ModesZM5.LMode.UpperLevelPLCAlarmA OR #IO_ModesZM5.LMode.UpperLevelPLCAlarmB) AND NOT #IO_ModesZM5.LMode.UpperLevelPLCAlarmABCondition) OR ((#IO_ModesZM6.LMode.UpperLevelPLCAlarmA OR #IO_ModesZM6.LMode.UpperLevelPLCAlarmB) AND NOT #IO_ModesZM6.LMode.UpperLevelPLCAlarmABCondition) OR ((#IO_ModesZM7.LMode.UpperLevelPLCAlarmA OR #IO_ModesZM7.LMode.UpperLevelPLCAlarmB) AND NOT #IO_ModesZM7.LMode.UpperLevelPLCAlarmABCondition) OR ((#IO_ModesZM8.LMode.UpperLevelPLCAlarmA OR #IO_ModesZM8.LMode.UpperLevelPLCAlarmB) AND NOT #IO_ModesZM8.LMode.UpperLevelPLCAlarmABCondition) OR ((#IO_ModesZM9.LMode.UpperLevelPLCAlarmA OR #IO_ModesZM9.LMode.UpperLevelPLCAlarmB) AND NOT #IO_ModesZM9.LMode.UpperLevelPLCAlarmABCondition) OR ((#IO_ModesZM10.LMode.UpperLevelPLCAlarmA OR #IO_ModesZM10.LMode.UpperLevelPLCAlarmB) AND NOT #IO_ModesZM10.LMode.UpperLevelPLCAlarmABCondition) OR ((#IO_ModesZM11.LMode.UpperLevelPLCAlarmA OR #IO_ModesZM11.LMode.UpperLevelPLCAlarmB) AND NOT #IO_ModesZM11.LMode.UpperLevelPLCAlarmABCondition) OR ((#IO_ModesZM12.LMode.UpperLevelPLCAlarmA OR #IO_ModesZM12.LMode.UpperLevelPLCAlarmB) AND NOT #IO_ModesZM12.LMode.UpperLevelPLCAlarmABCondition) OR ((#IO_ModesZM13.LMode.UpperLevelPLCAlarmA OR #IO_ModesZM13.LMode.UpperLevelPLCAlarmB) AND NOT #IO_ModesZM13.LMode.UpperLevelPLCAlarmABCondition) OR ((#IO_ModesZM14.LMode.UpperLevelPLCAlarmA OR #IO_ModesZM14.LMode.UpperLevelPLCAlarmB) AND NOT #IO_ModesZM14.LMode.UpperLevelPLCAlarmABCondition) OR ((#IO_ModesZM15.LMode.UpperLevelPLCAlarmA OR #IO_ModesZM15.LMode.UpperLevelPLCAlarmB) AND NOT #IO_ModesZM15.LMode.UpperLevelPLCAlarmABCondition) OR ((#IO_ModesZM16.LMode.UpperLevelPLCAlarmA OR #IO_ModesZM16.LMode.UpperLevelPLCAlarmB) AND NOT #IO_ModesZM16.LMode.UpperLevelPLCAlarmABCondition);
END_REGION

REGION Network 7: **** 4.2 - Machine status - Calculated **** Lamptest
   // Lamptest
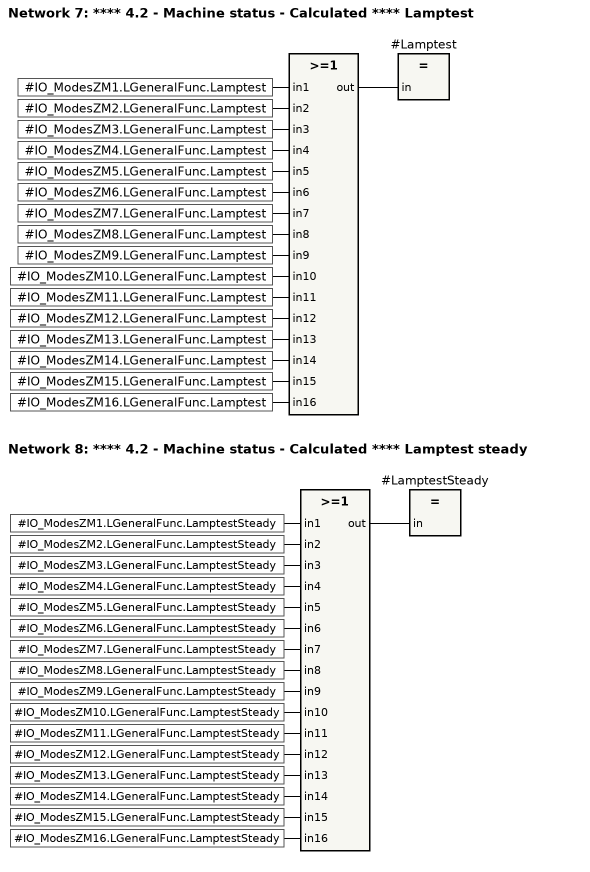
   #Lamptest := #IO_ModesZM1.LGeneralFunc.Lamptest OR #IO_ModesZM2.LGeneralFunc.Lamptest OR #IO_ModesZM3.LGeneralFunc.Lamptest OR #IO_ModesZM4.LGeneralFunc.Lamptest OR #IO_ModesZM5.LGeneralFunc.Lamptest OR #IO_ModesZM6.LGeneralFunc.Lamptest OR #IO_ModesZM7.LGeneralFunc.Lamptest OR #IO_ModesZM8.LGeneralFunc.Lamptest OR #IO_ModesZM9.LGeneralFunc.Lamptest OR #IO_ModesZM10.LGeneralFunc.Lamptest OR #IO_ModesZM11.LGeneralFunc.Lamptest OR #IO_ModesZM12.LGeneralFunc.Lamptest OR #IO_ModesZM13.LGeneralFunc.Lamptest OR #IO_ModesZM14.LGeneralFunc.Lamptest OR #IO_ModesZM15.LGeneralFunc.Lamptest OR #IO_ModesZM16.LGeneralFunc.Lamptest;
END_REGION

REGION Network 8: **** 4.2 - Machine status - Calculated **** Lamptest steady
   // Lamptest
   #LamptestSteady := #IO_ModesZM1.LGeneralFunc.LamptestSteady OR #IO_ModesZM2.LGeneralFunc.LamptestSteady OR #IO_ModesZM3.LGeneralFunc.LamptestSteady OR #IO_ModesZM4.LGeneralFunc.LamptestSteady OR #IO_ModesZM5.LGeneralFunc.LamptestSteady OR #IO_ModesZM6.LGeneralFunc.LamptestSteady OR #IO_ModesZM7.LGeneralFunc.LamptestSteady OR #IO_ModesZM8.LGeneralFunc.LamptestSteady OR #IO_ModesZM9.LGeneralFunc.LamptestSteady OR #IO_ModesZM10.LGeneralFunc.LamptestSteady OR #IO_ModesZM11.LGeneralFunc.LamptestSteady OR #IO_ModesZM12.LGeneralFunc.LamptestSteady OR #IO_ModesZM13.LGeneralFunc.LamptestSteady OR #IO_ModesZM14.LGeneralFunc.LamptestSteady OR #IO_ModesZM15.LGeneralFunc.LamptestSteady OR #IO_ModesZM16.LGeneralFunc.LamptestSteady;
END_REGION

REGION Network 9: **** 4.2 - Machine status - Calculated **** Automatic mode selected
   // Automatic mode selected
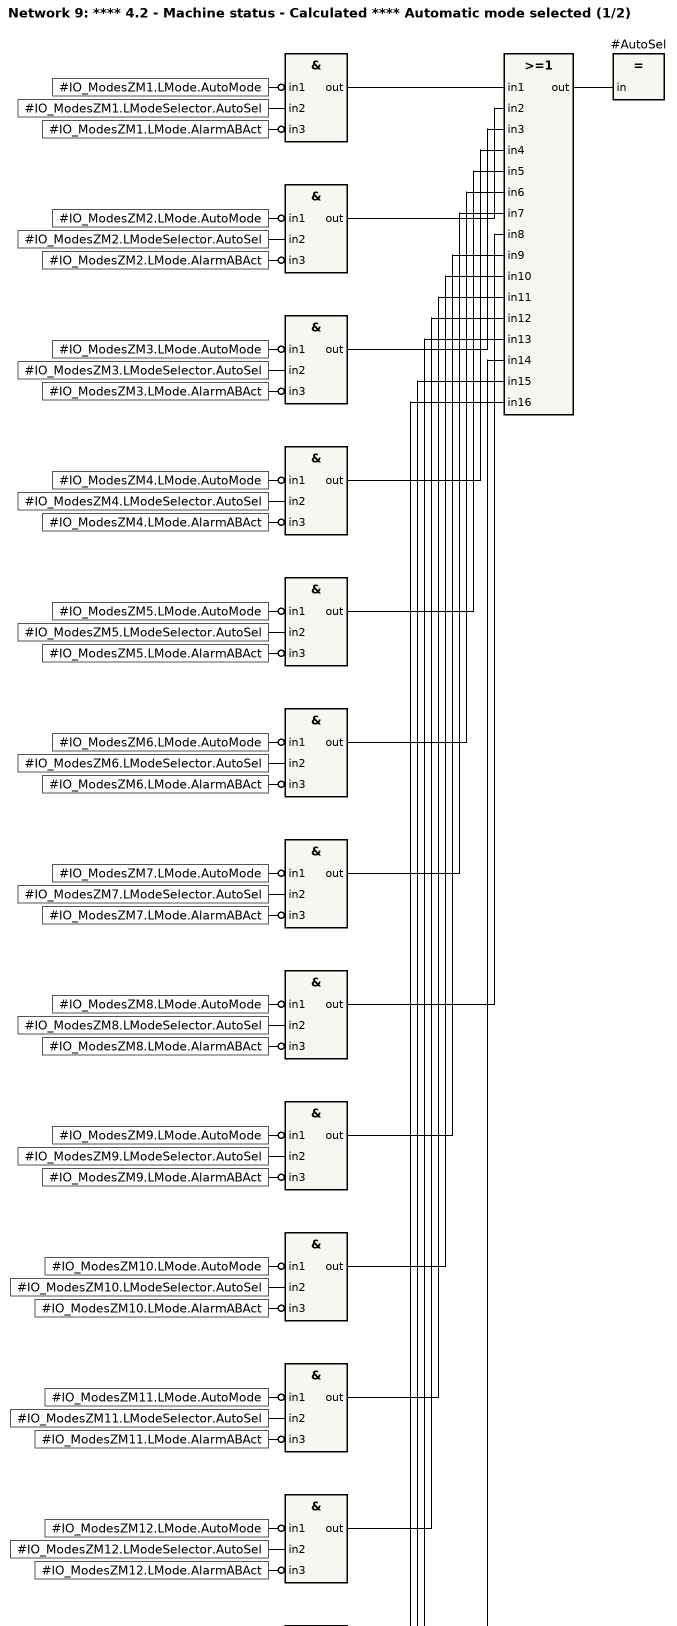
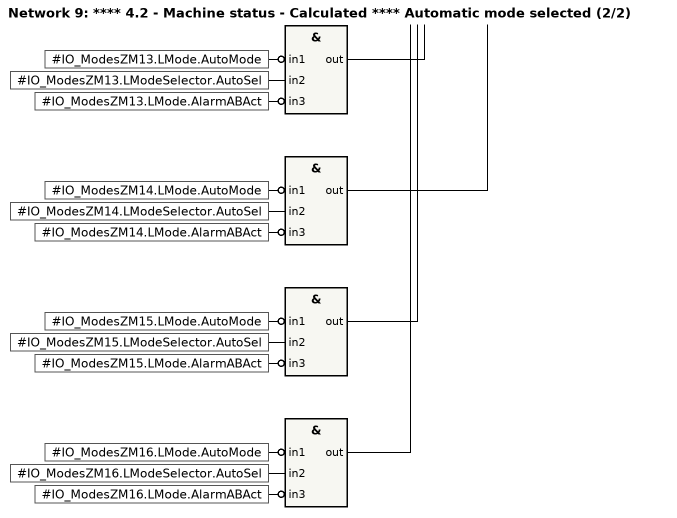
   #AutoSel := (NOT #IO_ModesZM1.LMode.AutoMode AND #IO_ModesZM1.LModeSelector.AutoSel AND NOT #IO_ModesZM1.LMode.AlarmABAct) OR (NOT #IO_ModesZM2.LMode.AutoMode AND #IO_ModesZM2.LModeSelector.AutoSel AND NOT #IO_ModesZM2.LMode.AlarmABAct) OR (NOT #IO_ModesZM3.LMode.AutoMode AND #IO_ModesZM3.LModeSelector.AutoSel AND NOT #IO_ModesZM3.LMode.AlarmABAct) OR (NOT #IO_ModesZM4.LMode.AutoMode AND #IO_ModesZM4.LModeSelector.AutoSel AND NOT #IO_ModesZM4.LMode.AlarmABAct) OR (NOT #IO_ModesZM5.LMode.AutoMode AND #IO_ModesZM5.LModeSelector.AutoSel AND NOT #IO_ModesZM5.LMode.AlarmABAct) OR (NOT #IO_ModesZM6.LMode.AutoMode AND #IO_ModesZM6.LModeSelector.AutoSel AND NOT #IO_ModesZM6.LMode.AlarmABAct) OR (NOT #IO_ModesZM7.LMode.AutoMode AND #IO_ModesZM7.LModeSelector.AutoSel AND NOT #IO_ModesZM7.LMode.AlarmABAct) OR (NOT #IO_ModesZM8.LMode.AutoMode AND #IO_ModesZM8.LModeSelector.AutoSel AND NOT #IO_ModesZM8.LMode.AlarmABAct) OR (NOT #IO_ModesZM9.LMode.AutoMode AND #IO_ModesZM9.LModeSelector.AutoSel AND NOT #IO_ModesZM9.LMode.AlarmABAct) OR (NOT #IO_ModesZM10.LMode.AutoMode AND #IO_ModesZM10.LModeSelector.AutoSel AND NOT #IO_ModesZM10.LMode.AlarmABAct) OR (NOT #IO_ModesZM11.LMode.AutoMode AND #IO_ModesZM11.LModeSelector.AutoSel AND NOT #IO_ModesZM11.LMode.AlarmABAct) OR (NOT #IO_ModesZM12.LMode.AutoMode AND #IO_ModesZM12.LModeSelector.AutoSel AND NOT #IO_ModesZM12.LMode.AlarmABAct) OR (NOT #IO_ModesZM13.LMode.AutoMode AND #IO_ModesZM13.LModeSelector.AutoSel AND NOT #IO_ModesZM13.LMode.AlarmABAct) OR (NOT #IO_ModesZM14.LMode.AutoMode AND #IO_ModesZM14.LModeSelector.AutoSel AND NOT #IO_ModesZM14.LMode.AlarmABAct) OR (NOT #IO_ModesZM15.LMode.AutoMode AND #IO_ModesZM15.LModeSelector.AutoSel AND NOT #IO_ModesZM15.LMode.AlarmABAct) OR (NOT #IO_ModesZM16.LMode.AutoMode AND #IO_ModesZM16.LModeSelector.AutoSel AND NOT #IO_ModesZM16.LMode.AlarmABAct);
END_REGION

REGION Network 10: **** 4.2 - Machine status - Calculated **** Automatic mode active
   // Automatic mode active
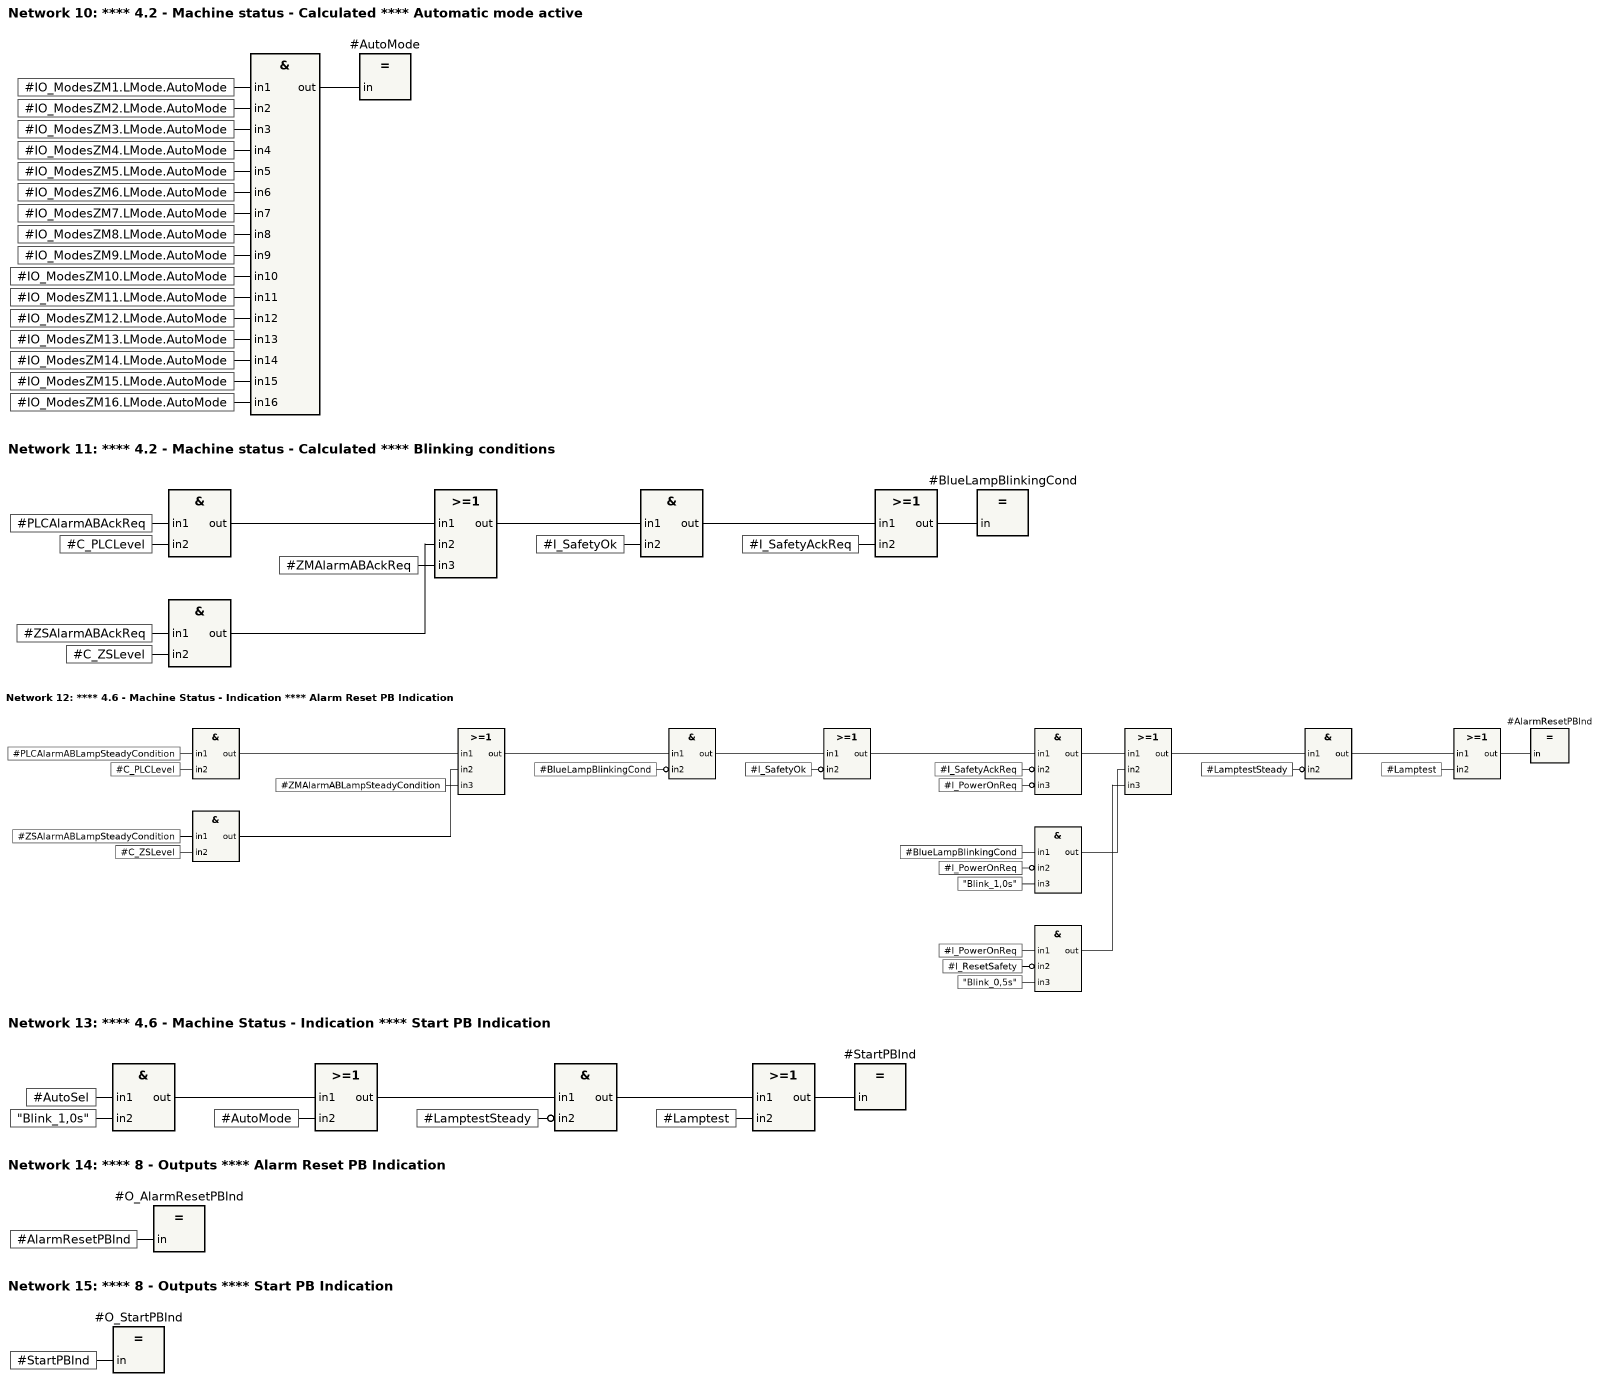
   #AutoMode := #IO_ModesZM1.LMode.AutoMode AND #IO_ModesZM2.LMode.AutoMode AND #IO_ModesZM3.LMode.AutoMode AND #IO_ModesZM4.LMode.AutoMode AND #IO_ModesZM5.LMode.AutoMode AND #IO_ModesZM6.LMode.AutoMode AND #IO_ModesZM7.LMode.AutoMode AND #IO_ModesZM8.LMode.AutoMode AND #IO_ModesZM9.LMode.AutoMode AND #IO_ModesZM10.LMode.AutoMode AND #IO_ModesZM11.LMode.AutoMode AND #IO_ModesZM12.LMode.AutoMode AND #IO_ModesZM13.LMode.AutoMode AND #IO_ModesZM14.LMode.AutoMode AND #IO_ModesZM15.LMode.AutoMode AND #IO_ModesZM16.LMode.AutoMode;
END_REGION

REGION Network 11: **** 4.2 - Machine status - Calculated **** Blinking conditions
   // Blinking conditions
   #BlueLampBlinkingCond := (((#PLCAlarmABAckReq AND #C_PLCLevel) OR (#ZSAlarmABAckReq AND #C_ZSLevel) OR #ZMAlarmABAckReq) AND #I_SafetyOk) OR #I_SafetyAckReq;
END_REGION

REGION Network 12: **** 4.6 - Machine Status - Indication **** Alarm Reset PB Indication
   // Alarm Reset PB indication
   #AlarmResetPBInd := (((((((#PLCAlarmABLampSteadyCondition AND #C_PLCLevel) OR (#ZSAlarmABLampSteadyCondition AND #C_ZSLevel) OR #ZMAlarmABLampSteadyCondition) AND NOT #BlueLampBlinkingCond) OR NOT #I_SafetyOk) AND NOT #I_SafetyAckReq AND NOT #I_PowerOnReq) OR (#BlueLampBlinkingCond AND NOT #I_PowerOnReq AND "Blink_1,0s") OR (#I_PowerOnReq AND NOT #I_ResetSafety AND "Blink_0,5s")) AND NOT #LamptestSteady) OR #Lamptest;
END_REGION

REGION Network 13: **** 4.6 - Machine Status - Indication **** Start PB Indication
   // Start PB indication
   #StartPBInd := (((#AutoSel AND "Blink_1,0s") OR #AutoMode) AND NOT #LamptestSteady) OR #Lamptest;
END_REGION

REGION Network 14: **** 8 - Outputs **** Alarm Reset PB Indication
   // Alarm Reset PB Indication
   #O_AlarmResetPBInd := #AlarmResetPBInd;
END_REGION

REGION Network 15: **** 8 - Outputs **** Start PB Indication
   // Start PB Indication
   #O_StartPBInd := #StartPBInd;
END_REGION
END_FUNCTION_BLOCK
